// TIA Portal V19 export
DATA_BLOCK "Config"   // DB72
// stored: Access Published, MemoryReserve 100, Namespace Unit2.EM2
   VAR
      em { ExternalWritable := 'False'} : "LAF_typeEmConfiguration";   // Configuration of EM Parameters
      axis { ExternalWritable := 'False'} : Array[1.._.U2EM2_NO_OF_AXES] of DB_ANY;   // Assign the axis of the EM
      em2Parameters : "LAF_typeConstraintRollerEm2Parameters";
   END_VAR
BEGIN
   em.referenceDesignator.parent := WSTRING#'U1';
   em.referenceDesignator.relative := WSTRING#'EM1';
   // em2Parameters.cm5Axis107.production.distanceList[0] : 24电芯 首位位置
   // em2Parameters.cm5Axis107.production.distanceList[1] : 24电芯末尾位位置
   // em2Parameters.cm5Axis107.production.distanceList[2] : 24 总长度 [1]-[0]
   // em2Parameters.cm5Axis107.production.distanceList[3] : 36电芯 首位位置
   // em2Parameters.cm5Axis107.production.distanceList[4] : 36电芯末尾位位置
   // em2Parameters.cm5Axis107.production.distanceList[5] : 36 总长度 [1]-[0]
   // em2Parameters.cm5Axis107.production.distanceList[6] : Structure for a Position set point
   // em2Parameters.cm5Axis107.production.distanceList[7] : Structure for a Position set point
   // em2Parameters.cm5Axis107.production.distanceList[8] : Structure for a Position set point
   // em2Parameters.cm5Axis107.production.distanceList[9] : Structure for a Position set point
   // em2Parameters.cm5Axis107.production.distanceList[10] : Structure for a Position set point
   // em2Parameters.cm5Axis107.production.distanceList[11] : Structure for a Position set point
   // em2Parameters.cm5Axis107.production.distanceList[12] : Structure for a Position set point
   // em2Parameters.cm5Axis107.production.distanceList[13] : Structure for a Position set point
   // em2Parameters.cm5Axis107.production.distanceList[14] : Structure for a Position set point
   // em2Parameters.cm5Axis107.production.distanceList[15] : Structure for a Position set point
   // em2Parameters.cm5Axis107.production.distanceList[16] : Structure for a Position set point
   // em2Parameters.cm5Axis107.production.distanceList[17] : Structure for a Position set point
   // em2Parameters.cm5Axis107.production.distanceList[18] : Structure for a Position set point
   // em2Parameters.cm5Axis107.production.distanceList[19] : Structure for a Position set point
   // em2Parameters.cm5Axis107.production.distanceList[20] : 24电芯 第一次顶位置
   // em2Parameters.cm5Axis107.production.distanceList[21] : 24电芯 第二次顶位置
   // em2Parameters.cm5Axis107.production.distanceList[22] : 24电芯 第三次顶位置
   // em2Parameters.cm5Axis107.production.distanceList[23] : Structure for a Position set point
   // em2Parameters.cm5Axis107.production.distanceList[24] : Structure for a Position set point
   // em2Parameters.cm5Axis107.production.distanceList[25] : Structure for a Position set point
   // em2Parameters.cm5Axis107.production.distanceList[26] : Structure for a Position set point
   // em2Parameters.cm5Axis107.production.distanceList[27] : Structure for a Position set point
   // em2Parameters.cm5Axis107.production.distanceList[28] : Structure for a Position set point
   // em2Parameters.cm5Axis107.production.distanceList[29] : Structure for a Position set point
   // em2Parameters.cm5Axis107.production.distanceList[30] : 36电芯 第一次顶位置
   // em2Parameters.cm5Axis107.production.distanceList[31] : 36电芯 第2次顶位置
   // em2Parameters.cm5Axis107.production.distanceList[32] : 36电芯 第3次顶位置
   // em2Parameters.cm5Axis107.production.distanceList[33] : 36电芯 第4次顶位置
   // em2Parameters.cm5Axis107.production.distanceList[34] : 36电芯 第5次顶位置
   em2Parameters.cm5Axis107.production.distanceList[0].position := 20.0;
   em2Parameters.cm5Axis107.production.distanceList[1].position := 140.0;
   em2Parameters.cm5Axis107.production.distanceList[3].position := 30.0;
   em2Parameters.cm5Axis107.production.distanceList[4].position := 210.0;
   em2Parameters.cm5Axis107.production.distanceList[0..1].velocity := 20.0;
   em2Parameters.cm5Axis107.production.distanceList[3..4].velocity := 30.0;
END_DATA_BLOCK
